(* IEC 61131-3 sources: Industry-PLC-LLM/data/PLCBEAD_repo/PLCBEAD_PLCEmbed-main/PLC-BEAD/Source/GEB/_WORD_TO_DINT, 1 file *)

(* ---- _WORD_TO_DINT.ST ---- *)
FUNCTION _WORD_TO_DINT:DINT
	VAR_INPUT
		IN :	WORD;
	END_VAR
	_WORD_TO_DINT := UINT_TO_DINT(WORD_TO_UINT(IN));
END_FUNCTION
PROGRAM program0
  VAR
    LocalVar0 : WORD;
    LocalOUT  : DINT;
  END_VAR

  LocalOUT := _WORD_TO_DINT(LocalVar0);
END_PROGRAM
